{attribute 'GeneratedUsingTerminal: AX8118-0100-0101-0101'}
{attribute addProperty BoxType "AX8118-0100-0101-0101"}
{attribute addProperty Id "DeviceDevice_6E2575772Device_SafetyDevice_Safety_C21945A160Ch_ACh_A_1FF86D8522WcStateAT %I*WcState_B516A2644InfoDataAT %I*InfoData_D1E293FD11"}
{attribute addProperty CRC "1656469377"}
{attribute addProperty Size "99"}
TYPE AX8118_62BBB781 EXTENDS EtcSlaveTerminalBase_947E5A46 :
STRUCT
	{attribute addProperty Name "Device"}
	Device : Device_6E257577;
	{attribute addProperty Name "Device_Safety"}
	Device_Safety : Device_Safety_C21945A1;
	{attribute addProperty Name "Ch_A"}
	Ch_A : Ch_A_1FF86D85;
	{attribute addProperty Name "WcState"}
	WcState : WcState_B516A264;
	{attribute addProperty Name "InfoData"}
	InfoData : InfoData_D1E293FD;
END_STRUCT
END_TYPE

(* stored: Version 1.2.0.0, ProductVersion 3.1.4024.9
   DUT AX8118_62BBB781: Id {b8d65c6b-c3a7-4d56-ae29-450433320155} *)
